ORGANIZATION_BLOCK OB 1
	VAR_TEMP
		RET_TMP		: INT;
		CDT_TMP		: DATE_AND_TIME;
	END_VAR
BEGIN
	CALL		SFC 1 (
		RET_VAL	:= #RET_TMP,
		CDT	:= #CDT_TMP,
	)
	__ASSERT==	__STW BIE,	1
	L		#RET_TMP
	__ASSERT==	__ACCU 1,	W#16#0000

	CALL SFC 46 // STOP CPU
END_ORGANIZATION_BLOCK
